TYPE ST_Trajectory :
STRUCT
	fPosition: LREAL;
	fVelocity: LREAL;
	fAcceleration: LREAL;
END_STRUCT
END_TYPE

(* stored: Version 1.1.0.1, ProductVersion 3.1.4024.5
   DUT ST_Trajectory: Id {62a5f936-2464-4b3c-a696-77b34f02ac89} *)
